// Mitsubishi GX Works2 project: e03   PLC: Q02/Q02H

PROGRAM MAIN
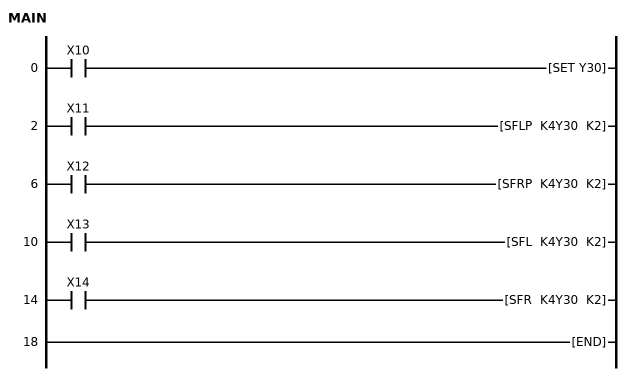
0     LD      X10
      SET     Y30
2     LD      X11
      SFLP    K4Y30 K2
6     LD      X12
      SFRP    K4Y30 K2
10    LD      X13
      SFL     K4Y30 K2
14    LD      X14
      SFR     K4Y30 K2
18    END
END_PROGRAM
